TYPE ST_MfcData :
STRUCT
	Addr : STRING(3); (* "@01".."@0A" *)
	Rfv : REAL; (* 현재 유량 *)
	Rfc : REAL; (* 현재 Set *)
	LastTx : STRING(128);
	LastRx : STRING(256);
	OkCnt : UDINT;
	ErrCnt : UDINT;
END_STRUCT
END_TYPE

(* stored: Version 1.1.0.1, ProductVersion 3.1.4024.15
   DUT ST_MfcData: Id {6a12b7e1-f253-4e25-bb12-c16cd1833c77} *)
